Staubli VAL3: AsynchStop.pgx

program AsynchStop()
begin
  //*******************************************************************************
  //*   ______
  //*  / _____) /|
  //* | |      / /
  //* | | /\  / /
  //* | | \ \/ /  _      Copyright (c) KEOLABS, 2016
  //* | |  \__/  | |        http://www.keolabs.com
  //* | |________| |
  //*  \__________/
  //*
  //********************************************************************************
  //*@file          : AsynchStop
  //*@author        : Yves Ragot
  //*@version       : $Id: AsynchStop.pgx 1365 2016-11-18 16:00:54Z yves $
  //*@brief         : Stop asynchronous mouvement
  //*
  //*******************************************************************************/

  // stop the mouvement
  stopMove()

  // clear all recorded commands
  if isEmpty() == false
    resetMotion()
  endIf

  // wait for mouvement ending
  waitEndMove()
  wait(isSettled())

  MoveRunning = false

end
